Fanuc KAREL source: kt00332.KL

-- PROVISIONAL review KL for V1013-1; original PC SHA256 d7b22583fa0138c1be338c48c2796521db22677c93a59533b78a3e5fee674e31
-- Incomplete behavior may be omitted. Consult companion uncertainty JSON. Do not deploy.
PROGRAM KT00332
%NOLOCKGROUP
VAR
  I1 : INTEGER
  OUT : BOOLEAN
-- UNRESOLVED_DECL H2 type=002017
BEGIN
  -- UNRESOLVED_PC offsets 5-16; opcodes 2E,23
  -- UNRESOLVED_PC offsets 21-35; opcodes 2E,22,9D,33,B4
  -- UNRESOLVED_PC offsets 40-62; opcodes 21,22,9D,33,B3,59,23
  -- UNRESOLVED_PC offsets 67-71; opcodes 7F
END KT00332
